// TIA Portal V18 export
// export: Created 2026-06-16T05:09:47.8032589Z, ExportSetting WithDefaults, DisplayName Totally Integrated Automation Portal, DisplayVersion V18 Update 5, DisplayName TIA Portal Openness, DisplayVersion V18 Update 5, DisplayName TIA Portal Version Control Interface, DisplayVersion V18, DisplayName SINAMICS Startdrive Advanced, DisplayVersion V18 SP2 Update 1, DisplayName SINAMICS Startdrive G110M, G120, G120C, G120D, G120P, G115D, DisplayVersion V18 SP2 Update 1, DisplayName SINAMICS Startdrive G130, G150, S120, S150, SINAMICS MV, S210, G220, S200, DisplayVersion V18 SP2 Update 1, DisplayName STEP 7 Professional, DisplayVersion V18 Update 5, DisplayName STEP 7 Safety, DisplayVersion V18, DisplayName WinCC Advanced / Unified PC, DisplayVersion V18 Update 5
FUNCTION "TEMPLATE--v1.0--07_Speed Control" : Void   // FC24, F_LAD
TITLE = Manage Safety Encoder
{ S7_Optimized_Access := 'TRUE' }
VERSION : 0.1
// v1.0 First Emission
// stored: AutoNumber true, IsIECCheckEnabled false, UDAEnableTagReadback false
BEGIN

REGION Network 1: !!NetworkComment$$
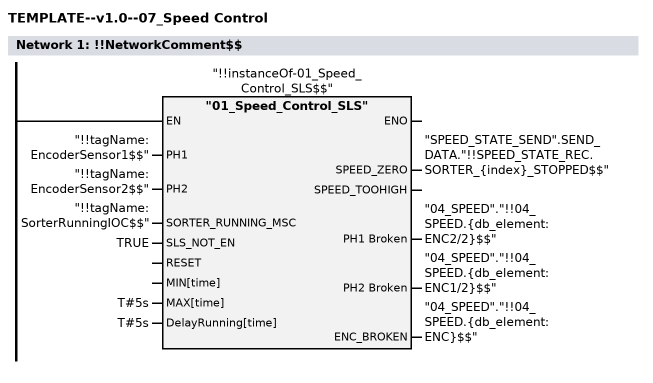
   RUNG wire#powerrail
      "!!instanceOf-01_Speed_Control_SLS$$"(PH1 := "!!tagName:EncoderSensor1$$", PH2 := "!!tagName:EncoderSensor2$$", SORTER_RUNNING_MSC := "!!tagName:SorterRunningIOC$$", SLS_NOT_EN := TRUE, RESET :=, "MIN[time]" :=, "MAX[time]" := T#5s, "DelayRunning[time]" := T#5s, SPEED_ZERO => "SPEED_STATE_SEND".SEND_DATA."!!SPEED_STATE_REC.SORTER_{index}_STOPPED$$", SPEED_TOOHIGH =>, "PH1 Broken" => "04_SPEED"."!!04_SPEED.{db_element:ENC2/2}$$", "PH2 Broken" => "04_SPEED"."!!04_SPEED.{db_element:ENC1/2}$$", ENC_BROKEN => "04_SPEED"."!!04_SPEED.{db_element:ENC}$$")
   END_RUNG
   // the same network as SCL:
   "!!instanceOf-01_Speed_Control_SLS$$"(PH1 := "!!tagName:EncoderSensor1$$",   // "01_Speed_Control_SLS"
                           PH2 := "!!tagName:EncoderSensor2$$",
                           SORTER_RUNNING_MSC := "!!tagName:SorterRunningIOC$$",
                           SLS_NOT_EN := TRUE,
                           "MAX[time]" := T#5s,
                           "DelayRunning[time]" := T#5s,
                           SPEED_ZERO => "SPEED_STATE_SEND".SEND_DATA."!!SPEED_STATE_REC.SORTER_{index}_STOPPED$$",
                           "PH1 Broken" => "04_SPEED"."!!04_SPEED.{db_element:ENC2/2}$$",
                           "PH2 Broken" => "04_SPEED"."!!04_SPEED.{db_element:ENC1/2}$$",
                           ENC_BROKEN => "04_SPEED"."!!04_SPEED.{db_element:ENC}$$");
END_REGION
END_FUNCTION
